TYPE ST_ACswitchgear_events :
STRUCT
	b_InputMCCBShuntFault	: BOOL;	
	b_OutputMCCBShuntFault	: BOOL;
	b_CEEprefuseFault		: BOOL;
	b_InputContactorFault	: BOOL;
END_STRUCT
END_TYPE

(* stored: Version 1.1.0.1, ProductVersion 3.1.4026.18
   DUT ST_ACswitchgear_events: Id {f040cb03-8bec-4ef8-8fa1-80f8f1fd17e3} *)
